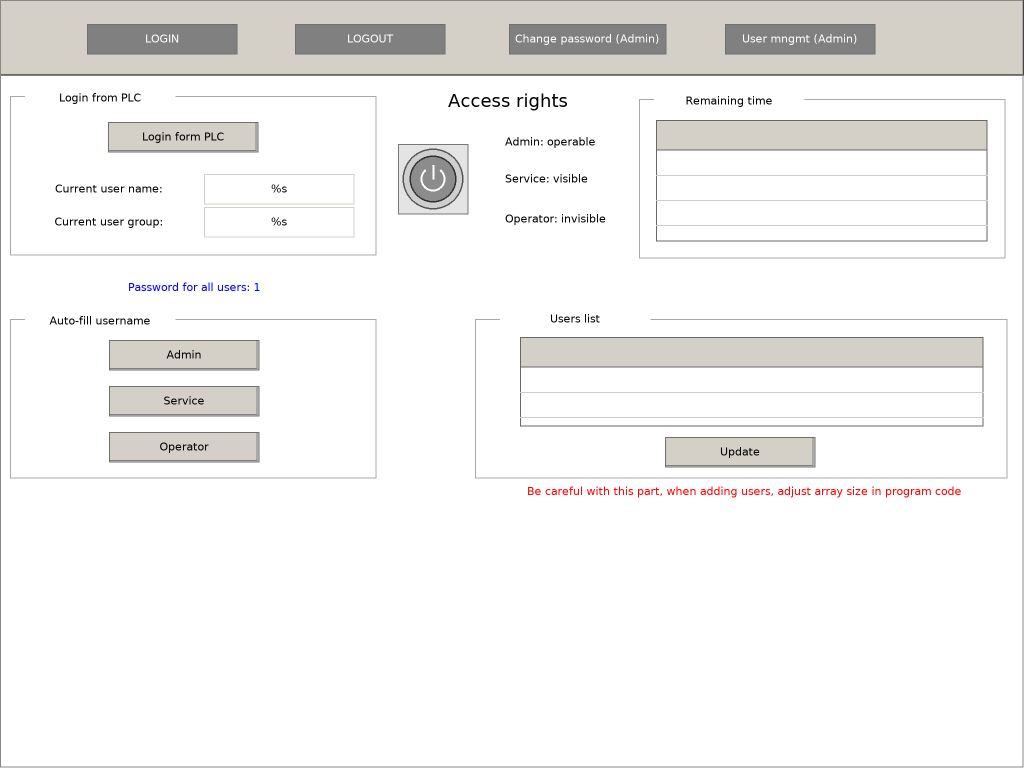
VISUALIZATION Visualization  // 1024x768
    Rectangle (10,319 366x159)
    Rectangle (639,99 366x159)
    Rectangle (0,0 1024x75)
    Button (87,24 150x30), "LOGIN"
        OnMouseDown: VisuUserMgmt Type=Login
    Button (295,24 150x30), "LOGOUT"
        OnMouseDown: VisuUserMgmt Type=Logout
    Button (509,24 157x30), "Change password (Admin)"
        OnMouseDown: VisuUserMgmt Type=ChangeUserPassword
    Button (725,24 150x30), "User mngmt (Admin)"
        OnMouseDown: VisuUserMgmt Type=OpenUserConfiguration
    Table (656,120 331x121), data array: P_TrackRemainingTime.aCurrentUser
        p3854506369: P_TrackRemainingTime.aCurrentUser[0,INDEX]
        p1892666644: P_TrackRemainingTime.aCurrentUser[1,INDEX]
        p338671338: P_TrackRemainingTime.aCurrentUser[2,INDEX]
        p2232123230: Name
        p511219082: Type
    Rectangle (654,86 150x30), "Remaining time"
    Rectangle (10,96 366x159)
    Rectangle (25,83 150x30), "Login from PLC"
    Button (108,122 150x30), "Login form PLC"
        tap P_LoginFromPLC.bLogIn
    Label (34,174 150x30), "Current user name:"
    Textfield (204,174 150x30), "%s", text variable: VisuElemsWinControls.CurrentUserName
    Rectangle (433,86 150x30), "Access rights"
    PowerSwitch (398,144 70x70), variable: MAIN.bButton, behaviour: TOGGLE, style: Switch-PowerSwitch-Gray
    Label (502,127 130x30), "Admin: operable"
    Label (502,164 130x30), "Service: visible"
    Label (502,204 130x30), "Operator: invisible"
    Rectangle (25,306 150x30), "Auto-fill username"
    Label (34,207 150x30), "Current user group:"
    Textfield (204,207 150x30), "%s", text variable: VisuElemsWinControls.CurrentUserGroupName
    Rectangle (475,319 532x159)
    Table (520,337 463x89), data array: P_ListUsers.aUsers
        p3854506369: P_ListUsers.aUsers[INDEX].wsUserName
        p1892666644: P_ListUsers.aUsers[INDEX].wsUserFullName
        p338671338: P_ListUsers.aUsers[INDEX].dwGroupID
        p2170511999: P_ListUsers.aUsers[INDEX].bDeactivated
        p511219082: Full Name
        p1755163831: Group ID
        p4092479075: Deactiated
    Rectangle (500,304 150x30), "Users list"
    Button (665,437 150x30), "Update"
        tap P_ListUsers.bUpdateUserList
    Label (483,463 523x57), "Be careful with this part, when adding users, adjust array size in program code"
    Label (13,259 363x57), "Password for all users: 1"
    Button (109,340 150x30), "Admin", colour toggle: VisuElemsWinControls.CurrentUserName="Admin"
        OnMouseDown: VisuUserMgmt Type=Login
        OnMouseDown: execute { VisuUserManagement.g_VisuLoginProviderManager.m_arrLoginProvider[0].stUserName := "Admin"; }
    Button (109,386 150x30), "Service", colour toggle: VisuElemsWinControls.CurrentUserName="Service"
        OnMouseDown: VisuUserMgmt Type=Login
        OnMouseDown: execute { VisuUserManagement.g_VisuLoginProviderManager.m_arrLoginProvider[0].stUserName := "Service"; }
    Button (109,432 150x30), "Operator", colour toggle: VisuElemsWinControls.CurrentUserName="Operator"
        OnMouseDown: VisuUserMgmt Type=Login
        OnMouseDown: execute { VisuUserManagement.g_VisuLoginProviderManager.m_arrLoginProvider[0].stUserName := "Operator"; }
END_VISUALIZATION

(* stored: Version 1.1.0.1, ProductVersion 3.1.4024.3
   Visu Visualization: Id {d3ce8fc7-b113-497a-bf46-bf0f08315645} *)
